// TIA Portal V20 export
FUNCTION "Service_ModuleService" : Void   // FC18, FBD
TITLE = Service
{ S7_Optimized_Access := 'TRUE' }
AUTHOR : Siemens AG
FAMILY : ServiceControl
VERSION : 1.0
// stored: SetENOAutomatically false
   VAR_TEMP
      ProcedureDone : Bool;
      UnholdingDone : Bool;
      StartingState : Bool;
      CompletingState : Bool;
      PausingState : Bool;
      HoldingState : Bool;
      AbortingState : Bool;
      StoppingState : Bool;
   END_VAR
BEGIN

REGION Network 1: Service
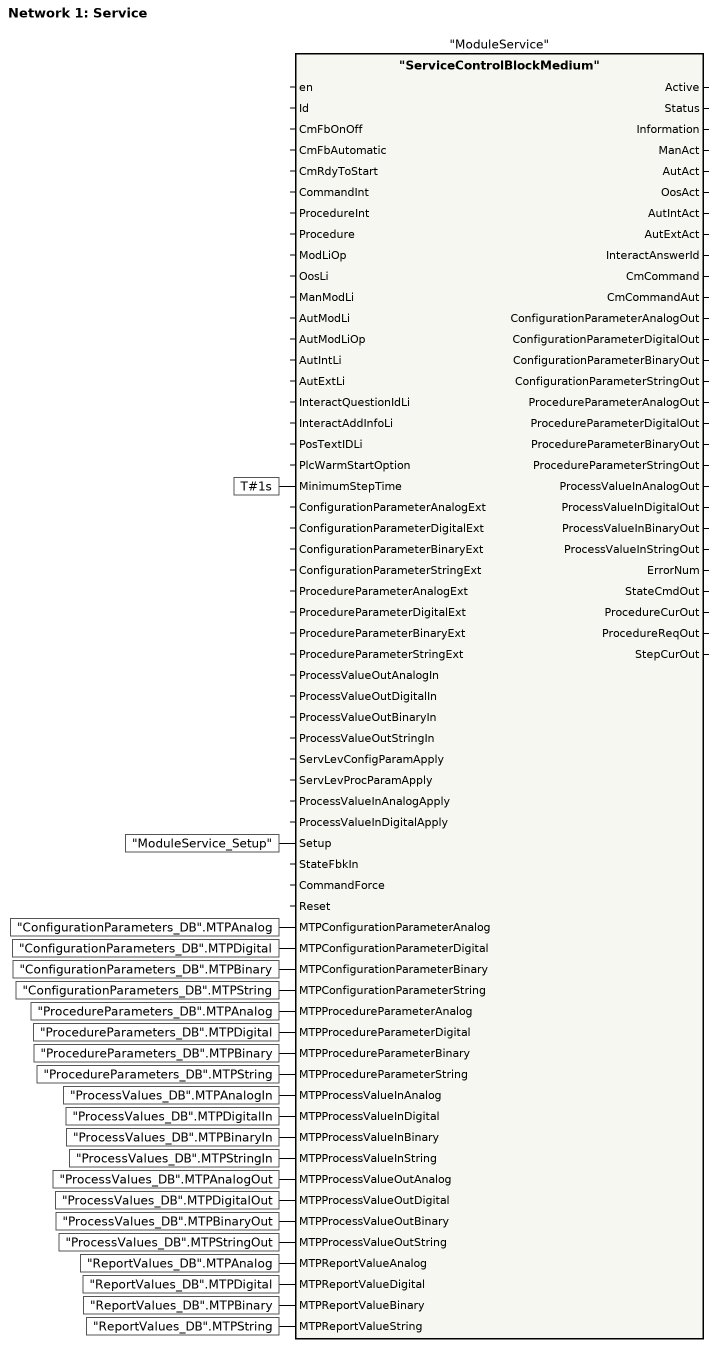
   "ModuleService"(MinimumStepTime := T#1s,   // "ServiceControlBlockMedium"
                   Setup := "ModuleService_Setup",
                   MTPConfigurationParameterAnalog := "ConfigurationParameters_DB".MTPAnalog,
                   MTPConfigurationParameterDigital := "ConfigurationParameters_DB".MTPDigital,
                   MTPConfigurationParameterBinary := "ConfigurationParameters_DB".MTPBinary,
                   MTPConfigurationParameterString := "ConfigurationParameters_DB".MTPString,
                   MTPProcedureParameterAnalog := "ProcedureParameters_DB".MTPAnalog,
                   MTPProcedureParameterDigital := "ProcedureParameters_DB".MTPDigital,
                   MTPProcedureParameterBinary := "ProcedureParameters_DB".MTPBinary,
                   MTPProcedureParameterString := "ProcedureParameters_DB".MTPString,
                   MTPProcessValueInAnalog := "ProcessValues_DB".MTPAnalogIn,
                   MTPProcessValueInDigital := "ProcessValues_DB".MTPDigitalIn,
                   MTPProcessValueInBinary := "ProcessValues_DB".MTPBinaryIn,
                   MTPProcessValueInString := "ProcessValues_DB".MTPStringIn,
                   MTPProcessValueOutAnalog := "ProcessValues_DB".MTPAnalogOut,
                   MTPProcessValueOutDigital := "ProcessValues_DB".MTPDigitalOut,
                   MTPProcessValueOutBinary := "ProcessValues_DB".MTPBinaryOut,
                   MTPProcessValueOutString := "ProcessValues_DB".MTPStringOut,
                   MTPReportValueAnalog := "ReportValues_DB".MTPAnalog,
                   MTPReportValueDigital := "ReportValues_DB".MTPDigital,
                   MTPReportValueBinary := "ReportValues_DB".MTPBinary,
                   MTPReportValueString := "ReportValues_DB".MTPString);
END_REGION

REGION Network 2: Service HMI
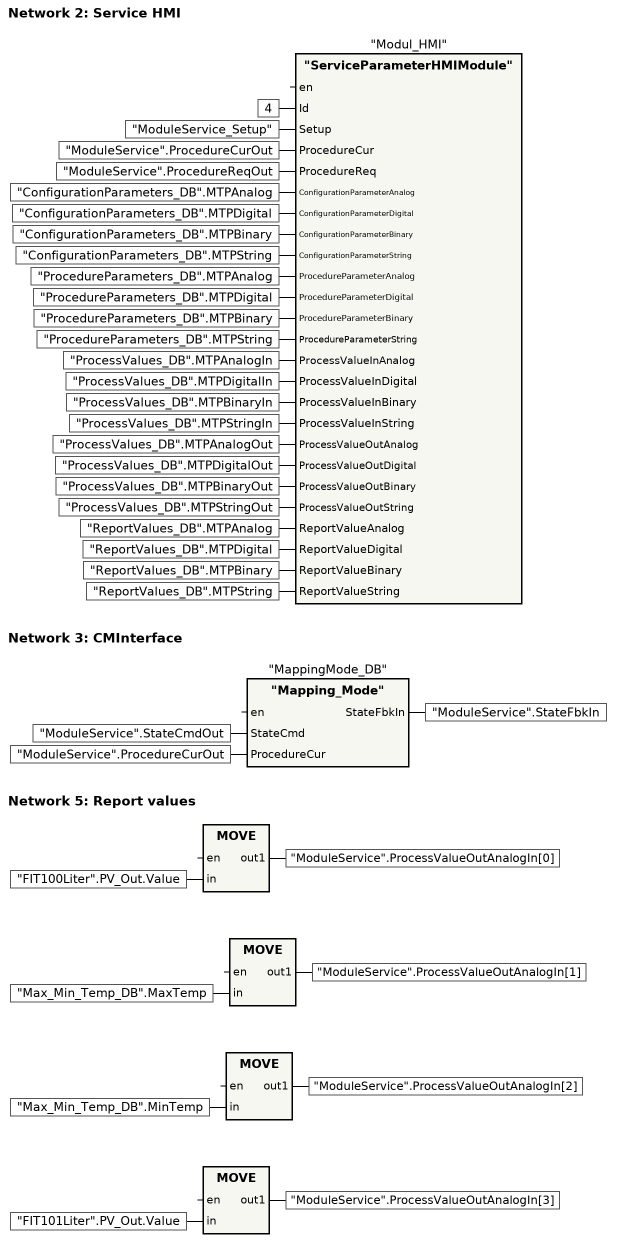
   "Modul_HMI"(Id := 4,   // "ServiceParameterHMIModule"
               Setup := "ModuleService_Setup",
               ProcedureCur := "ModuleService".ProcedureCurOut,
               ProcedureReq := "ModuleService".ProcedureReqOut,
               ConfigurationParameterAnalog := "ConfigurationParameters_DB".MTPAnalog,
               ConfigurationParameterDigital := "ConfigurationParameters_DB".MTPDigital,
               ConfigurationParameterBinary := "ConfigurationParameters_DB".MTPBinary,
               ConfigurationParameterString := "ConfigurationParameters_DB".MTPString,
               ProcedureParameterAnalog := "ProcedureParameters_DB".MTPAnalog,
               ProcedureParameterDigital := "ProcedureParameters_DB".MTPDigital,
               ProcedureParameterBinary := "ProcedureParameters_DB".MTPBinary,
               ProcedureParameterString := "ProcedureParameters_DB".MTPString,
               ProcessValueInAnalog := "ProcessValues_DB".MTPAnalogIn,
               ProcessValueInDigital := "ProcessValues_DB".MTPDigitalIn,
               ProcessValueInBinary := "ProcessValues_DB".MTPBinaryIn,
               ProcessValueInString := "ProcessValues_DB".MTPStringIn,
               ProcessValueOutAnalog := "ProcessValues_DB".MTPAnalogOut,
               ProcessValueOutDigital := "ProcessValues_DB".MTPDigitalOut,
               ProcessValueOutBinary := "ProcessValues_DB".MTPBinaryOut,
               ProcessValueOutString := "ProcessValues_DB".MTPStringOut,
               ReportValueAnalog := "ReportValues_DB".MTPAnalog,
               ReportValueDigital := "ReportValues_DB".MTPDigital,
               ReportValueBinary := "ReportValues_DB".MTPBinary,
               ReportValueString := "ReportValues_DB".MTPString);
END_REGION

REGION Network 3: CMInterface
   "MappingMode_DB"(StateCmd := "ModuleService".StateCmdOut,   // "Mapping_Mode"
                    ProcedureCur := "ModuleService".ProcedureCurOut,
                    StateFbkIn => "ModuleService".StateFbkIn);
END_REGION

REGION Network 4: Block pause and hold state
END_REGION

REGION Network 5: Report values
   "ModuleService".ProcessValueOutAnalogIn[0] := "FIT100Liter".PV_Out.Value;
   "ModuleService".ProcessValueOutAnalogIn[1] := "Max_Min_Temp_DB".MaxTemp;
   "ModuleService".ProcessValueOutAnalogIn[2] := "Max_Min_Temp_DB".MinTemp;
   "ModuleService".ProcessValueOutAnalogIn[3] := "FIT101Liter".PV_Out.Value;
END_REGION
END_FUNCTION
